(* Logix 5000 project; controller STAT 1756-L72 rev 20.12; software revision 20.04; part 33 of 34 *)
(* tags used below, declared in another part *)
   B3 : DINT[50];
   F8 : REAL[200];
   I1_000_Bit00 : ALIAS FOR stock:1:I.Point_0;   // disjoncteur algemeen
   I1_000_Bit01 : ALIAS FOR stock:1:I.Point_1;   // alim rechauffeur1
   I1_000_Bit02 : ALIAS FOR stock:1:I.Point_2;   // alim rechauffeur2
   I1_000_Bit03 : ALIAS FOR stock:1:I.Point_3;   // alim rechauffeur 3
   I1_000_Bit04 : ALIAS FOR stock:1:I.Point_4;   // alim rechauffeur 4
   I1_000_Bit05 : ALIAS FOR stock:1:I.Point_5;   // alim rechauffeur 5
   I1_000_Bit06 : ALIAS FOR stock:1:I.Point_6;   // protection pompesoude
   I1_000_Bit07 : ALIAS FOR stock:1:I.Point_7;   // protection pmp 2 acide
   I1_000_Bit08 : ALIAS FOR stock:1:I.Point_8;   // protection pmp acide
   I1_000_Bit15 : ALIAS FOR stock:1:I.Point_15;   // arret urgence
   I1_001_Bit09 : ALIAS FOR stock:1:I.Point_25;   // select.pmp soude sur drive
   I1_001_Bit11 : ALIAS FOR stock:1:I.Point_27;   // fault drivepmp soude
   I2_000_Bit00 : ALIAS FOR stock:2:I.Point_0;   // detection fuite soud
   I2_000_Bit01 : ALIAS FOR stock:2:I.Point_1;   // detection fuite acid
   I2_000_Bit02 : ALIAS FOR stock:2:I.Point_2;   // detection fuite mazo
   I2_000_Bit03 : ALIAS FOR stock:2:I.Point_3;   // wegskraan soude open
   I2_000_Bit04 : ALIAS FOR stock:2:I.Point_4;   // wegskraan soude dich
   I2_000_Bit07 : ALIAS FOR stock:2:I.Point_7;   // overfill stockagesoude
   I2_000_Bit08 : ALIAS FOR stock:2:I.Point_8;   // detection acideencuvement
   I2_000_Bit09 : ALIAS FOR stock:2:I.Point_9;   // detection soudeencuvement
   I2_000_Bit10 : ALIAS FOR stock:2:I.Point_10;   // fv vannesecuriteacide OUVERT
   I2_000_Bit11 : ALIAS FOR stock:2:I.Point_11;   // fv vannesecuriteacide FERME
   I2_001_Bit00 : ALIAS FOR stock:2:I.Point_16;   // NAOHL1 VA4FC O
   I2_001_Bit01 : ALIAS FOR stock:2:I.Point_17;   // NAOHL1 VA4FC F
   I2_001_Bit02 : ALIAS FOR stock:2:I.Point_18;   // NAOHL2 VA4FC O
   I2_001_Bit03 : ALIAS FOR stock:2:I.Point_19;   // NAOHL2 VA4FC O
   I2_001_Bit15 : ALIAS FOR stock:2:I.Point_31;   // pulse 0.1L passé
   N20 : DINT[100];
   N7 : DINT[255];
   O3_000_Bit00 : ALIAS FOR stock:3:O.Point_0;   // pompe soude
   O3_000_Bit08 : ALIAS FOR stock:3:O.Point_8;   // vanne soude
   O3_000_Bit09 : ALIAS FOR stock:3:O.Point_9;   // vannesecuriteacide
   O3_001_Bit11 : ALIAS FOR stock:3:O.Point_27;   // L1 VA4
   O3_001_Bit12 : ALIAS FOR stock:3:O.Point_28;   // NAOHL2 VA4
   T4 : TIMER[50];
   DateTime : DINT[7];   // DINT array tag for retrieve wallclock time through GSV created during conversion
   dmd_h2so4_ibt_ok : BOOL;
   dmd_soude_ibt_ok : BOOL;
   h2so4_ibt_finit : BOOL;
   I19_001_Bit05 : ALIAS FOR I19[1].5;   // vanne acide de stock fermee
   I19_001_Bit06 : ALIAS FOR I19[1].6;   // vanne acide de stock ouverte
   L1_stat : DINT[20];
   L2_STAT : DINT[20];
   L3_STAT : DINT[20];
   lancystock1 : DINT;
   lastmonth_h2so4_L1 : DINT;
   lastmonth_h2so4_L2 : DINT;
   lastmonth_h2so4_L3 : DINT;
   lastmonth_h2so4_L4 : DINT;
   lastmonth_h2so4_stat : REAL;
   lastmonth_naoh_L1 : DINT;
   lastmonth_naoh_L2 : DINT;
   lastmonth_naoh_L3 : DINT;
   lastmonth_naoh_L4 : DINT;
   lastmonth_naoh_stat : DINT;
   memo_flow_l1 : REAL;
   memo_flow_l2 : REAL;
   memo_flow_l3 : REAL;
   MW1 : BOOL;
   N : INT[255];
   O16_000_Bit03 : ALIAS FOR O16[0].3;
   ONS1 : DINT;
   passage_jourmois : BOOL;
   s_dmd_acid_ibt : DINT;
   S_dmd_naoh_ibt : REAL;
   s_lastmonth_tot_h2o_l1 : REAL;
   s_lastmonth_tot_h2o_l2 : REAL;
   s_lastmonth_tot_h2o_l3 : REAL;
   S_stock_v_h2so4_f : BOOL;
   S_stock_v_h2so4_o : BOOL;
   stat_L1 : DINT[20];
   STAT_L2 : DINT[20];
   STAT_L3 : DINT[20];
   stocklancy1 : DINT;
   stocklancy2 : DINT;
   tot_h2so4_stat : REAL;
   water_flow_to_l1 : REAL;
   water_flow_to_l2 : REAL;
   water_flow_to_l3 : REAL;
(* stock, continued *)

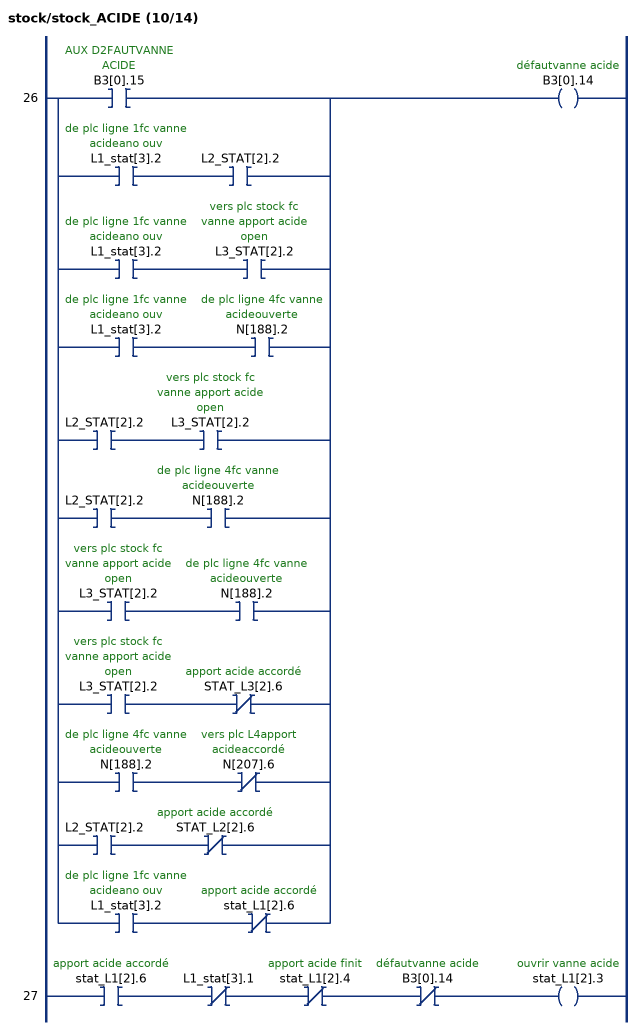
   [picture p674: stock/stock_ACIDE rungs 26-27]
   26: [XIC(B3[0].15) ,XIC(L1_stat[3].2) XIC(L2_STAT[2].2) ,XIC(L1_stat[3].2) XIC(L3_STAT[2].2) ,XIC(L1_stat[3].2) XIC(N[188].2) ,XIC(L2_STAT[2].2) XIC(L3_STAT[2].2) ,XIC(L2_STAT[2].2) XIC(N[188].2) ,XIC(L3_STAT[2].2) XIC(N[188].2) ,XIC(L3_STAT[2].2) XIO(STAT_L3[2].6) ,XIC(N[188].2) XIO(N[207].6) ,XIC(L2_STAT[2].2) XIO(STAT_L2[2].6) ,XIC(L1_stat[3].2) XIO(stat_L1[2].6) ]OTE(B3[0].14);
   27: XIC(stat_L1[2].6)XIO(L1_stat[3].1)XIO(stat_L1[2].4)XIO(B3[0].14)OTE(stat_L1[2].3);
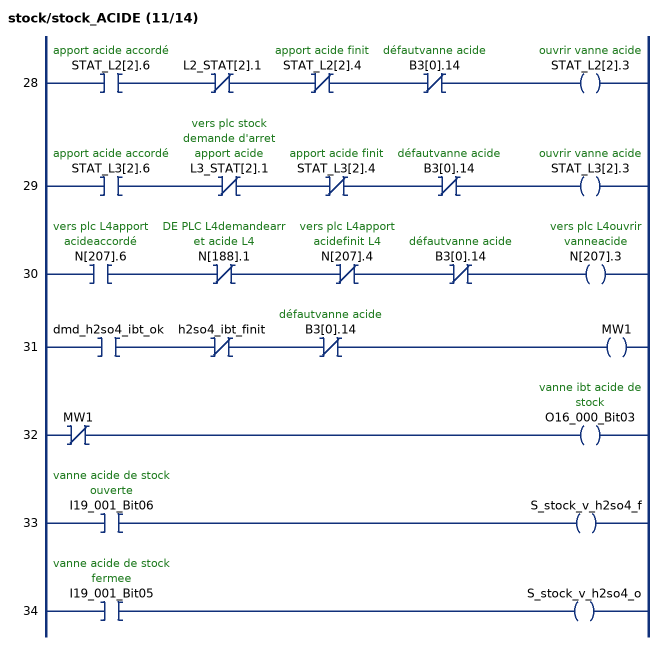
   28: XIC(STAT_L2[2].6)XIO(L2_STAT[2].1)XIO(STAT_L2[2].4)XIO(B3[0].14)OTE(STAT_L2[2].3);
   29: XIC(STAT_L3[2].6)XIO(L3_STAT[2].1)XIO(STAT_L3[2].4)XIO(B3[0].14)OTE(STAT_L3[2].3);
   30: XIC(N[207].6)XIO(N[188].1)XIO(N[207].4)XIO(B3[0].14)OTE(N[207].3);
   31: XIC(dmd_h2so4_ibt_ok)XIO(h2so4_ibt_finit)XIO(B3[0].14)OTE(MW1);
   32: XIO(MW1)OTE(O16_000_Bit03);
   33: XIC(I19_001_Bit06)OTE(S_stock_v_h2so4_f);
   34: XIC(I19_001_Bit05)OTE(S_stock_v_h2so4_o);
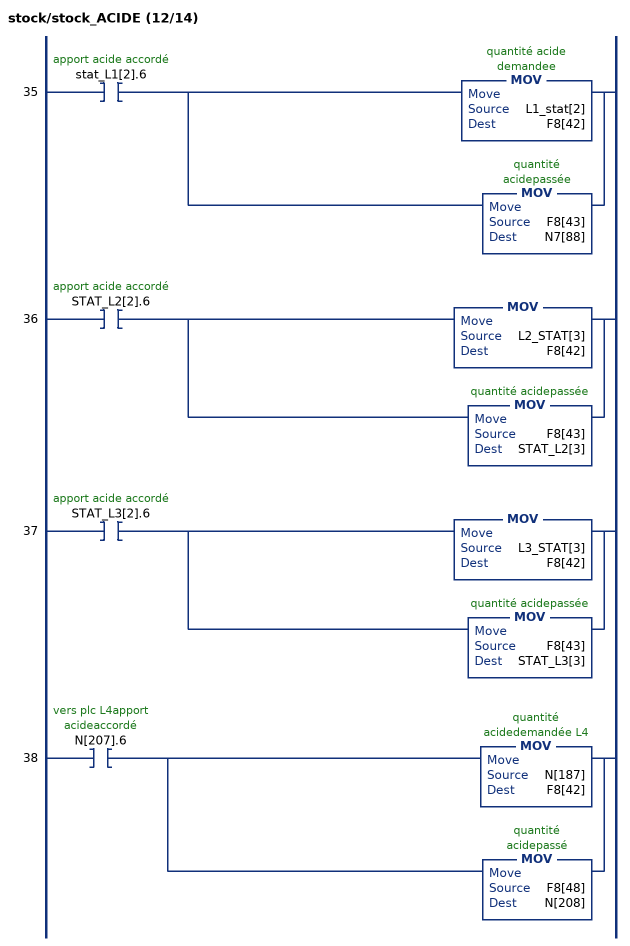
   35: XIC(stat_L1[2].6)[MOV(L1_stat[2],F8[42]) ,MOV(F8[43],N7[88]) ];
   36: XIC(STAT_L2[2].6)[MOV(L2_STAT[3],F8[42]) ,MOV(F8[43],STAT_L2[3]) ];
   37: XIC(STAT_L3[2].6)[MOV(L3_STAT[3],F8[42]) ,MOV(F8[43],STAT_L3[3]) ];
   38: XIC(N[207].6)[MOV(N[187],F8[42]) ,MOV(F8[48],N[208]) ];
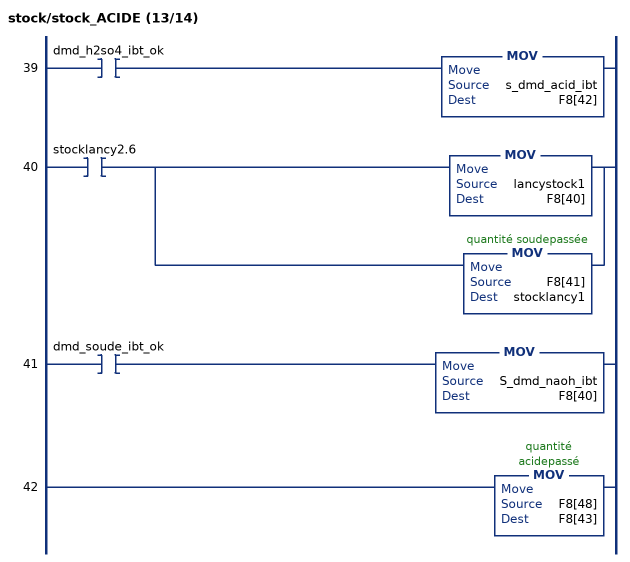
   39: XIC(dmd_h2so4_ibt_ok)MOV(s_dmd_acid_ibt,F8[42]);
   40: XIC(stocklancy2.6)[MOV(lancystock1,F8[40]) ,MOV(F8[41],stocklancy1) ];
   41: XIC(dmd_soude_ibt_ok)MOV(S_dmd_naoh_ibt,F8[40]);
   42: MOV(F8[48],F8[43]);
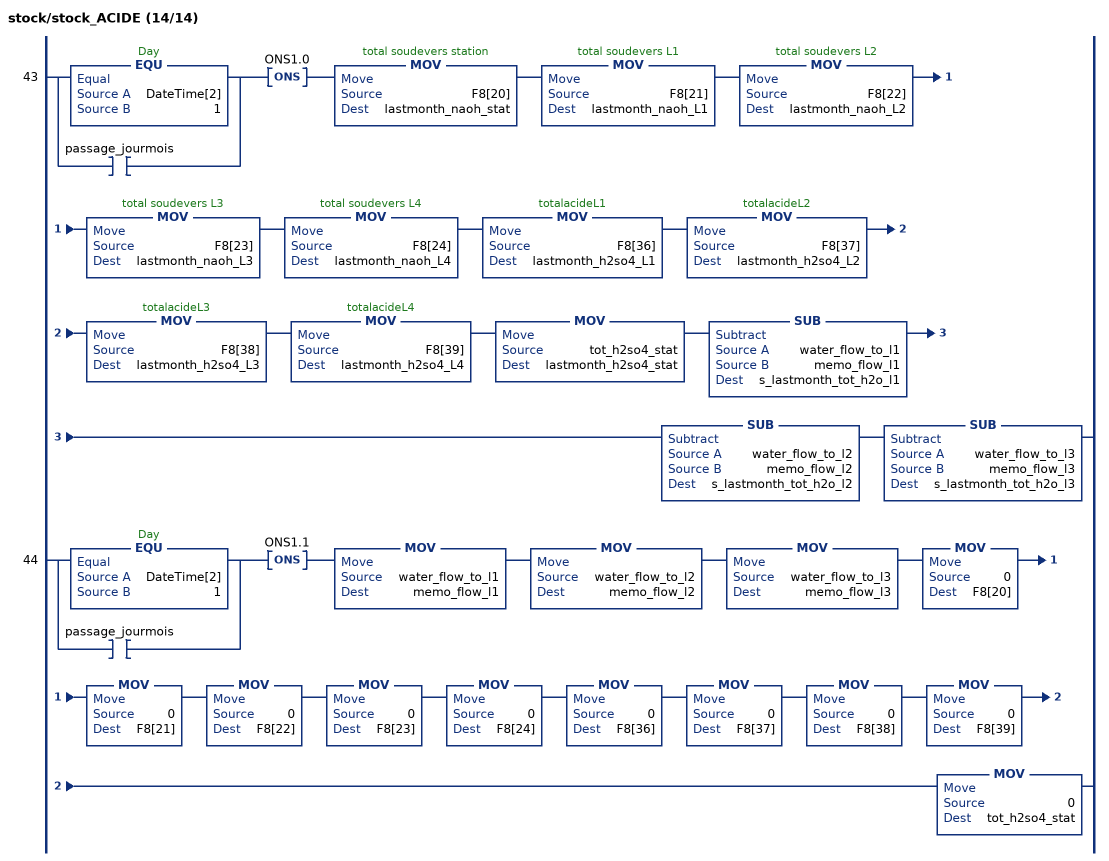
   43: [EQU(DateTime[2],1) ,XIC(passage_jourmois) ]ONS(ONS1.0)MOV(F8[20],lastmonth_naoh_stat)MOV(F8[21],lastmonth_naoh_L1)MOV(F8[22],lastmonth_naoh_L2)MOV(F8[23],lastmonth_naoh_L3)MOV(F8[24],lastmonth_naoh_L4)MOV(F8[36],lastmonth_h2so4_L1)MOV(F8[37],lastmonth_h2so4_L2)MOV(F8[38],lastmonth_h2so4_L3)MOV(F8[39],lastmonth_h2so4_L4)MOV(tot_h2so4_stat,lastmonth_h2so4_stat)SUB(water_flow_to_l1,memo_flow_l1,s_lastmonth_tot_h2o_l1)SUB(water_flow_to_l2,memo_flow_l2,s_lastmonth_tot_h2o_l2)SUB(water_flow_to_l3,memo_flow_l3,s_lastmonth_tot_h2o_l3);
   44: [EQU(DateTime[2],1) ,XIC(passage_jourmois) ]ONS(ONS1.1)MOV(water_flow_to_l1,memo_flow_l1)MOV(water_flow_to_l2,memo_flow_l2)MOV(water_flow_to_l3,memo_flow_l3)MOV(0,F8[20])MOV(0,F8[21])MOV(0,F8[22])MOV(0,F8[23])MOV(0,F8[24])MOV(0,F8[36])MOV(0,F8[37])MOV(0,F8[38])MOV(0,F8[39])MOV(0,tot_h2so4_stat);
END_ROUTINE

ROUTINE stock_ALARMING   (* ladder *)
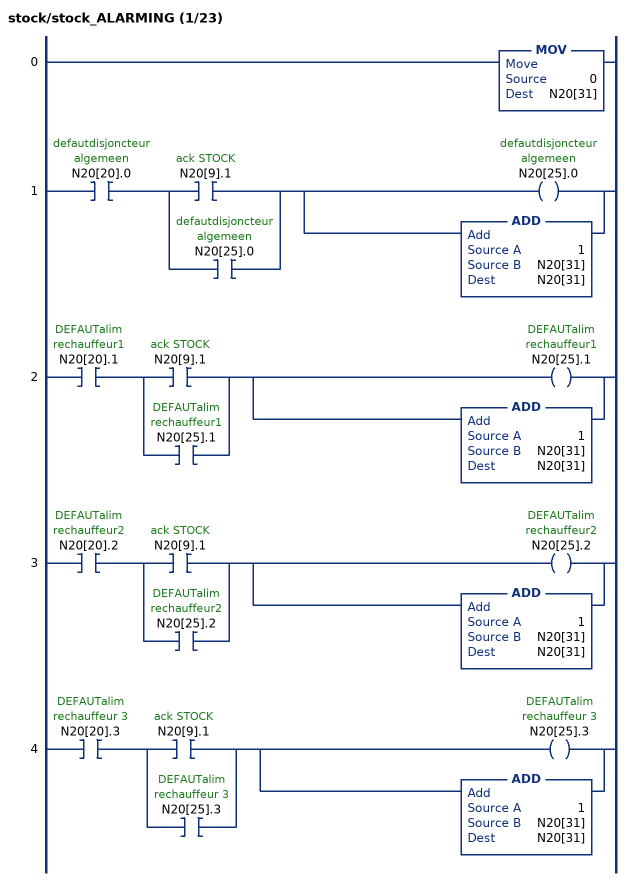
   0: MOV(0,N20[31]);
   1: XIC(N20[20].0)[XIC(N20[9].1) ,XIC(N20[25].0) ][OTE(N20[25].0) ,ADD(1,N20[31],N20[31]) ];
   2: XIC(N20[20].1)[XIC(N20[9].1) ,XIC(N20[25].1) ][OTE(N20[25].1) ,ADD(1,N20[31],N20[31]) ];
   3: XIC(N20[20].2)[XIC(N20[9].1) ,XIC(N20[25].2) ][OTE(N20[25].2) ,ADD(1,N20[31],N20[31]) ];
   4: XIC(N20[20].3)[XIC(N20[9].1) ,XIC(N20[25].3) ][OTE(N20[25].3) ,ADD(1,N20[31],N20[31]) ];
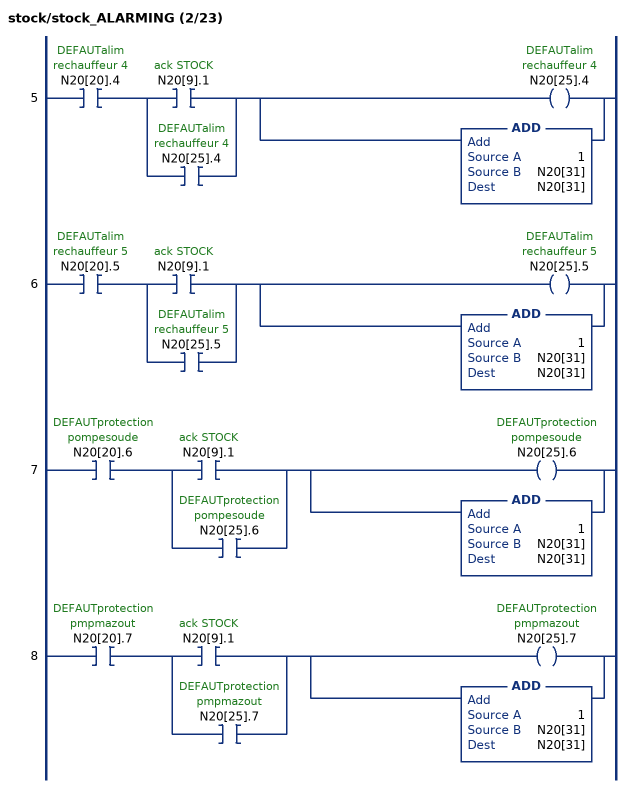
   5: XIC(N20[20].4)[XIC(N20[9].1) ,XIC(N20[25].4) ][OTE(N20[25].4) ,ADD(1,N20[31],N20[31]) ];
   6: XIC(N20[20].5)[XIC(N20[9].1) ,XIC(N20[25].5) ][OTE(N20[25].5) ,ADD(1,N20[31],N20[31]) ];
   7: XIC(N20[20].6)[XIC(N20[9].1) ,XIC(N20[25].6) ][OTE(N20[25].6) ,ADD(1,N20[31],N20[31]) ];
   8: XIC(N20[20].7)[XIC(N20[9].1) ,XIC(N20[25].7) ][OTE(N20[25].7) ,ADD(1,N20[31],N20[31]) ];
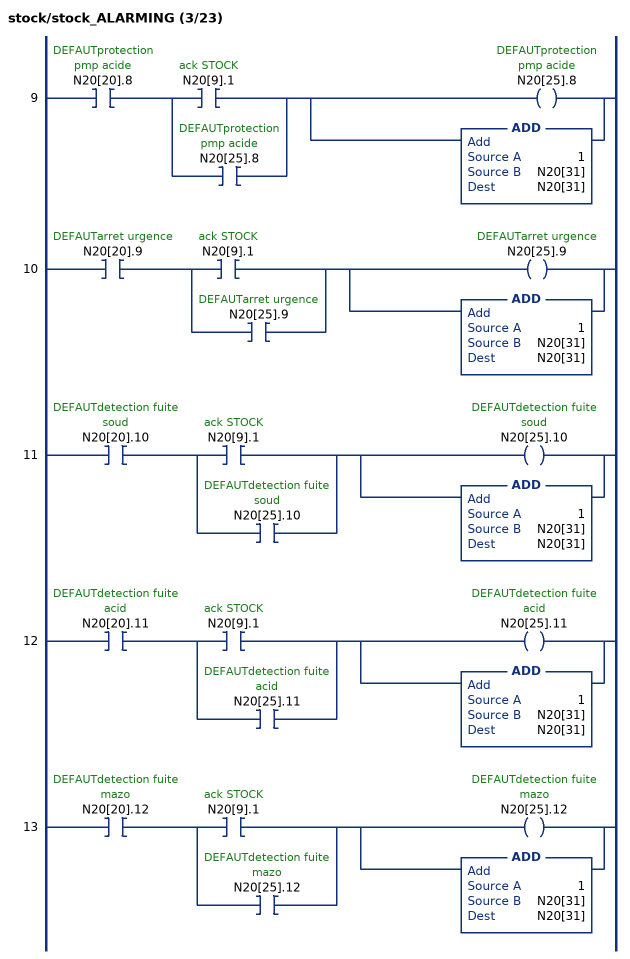
   9: XIC(N20[20].8)[XIC(N20[9].1) ,XIC(N20[25].8) ][OTE(N20[25].8) ,ADD(1,N20[31],N20[31]) ];
   10: XIC(N20[20].9)[XIC(N20[9].1) ,XIC(N20[25].9) ][OTE(N20[25].9) ,ADD(1,N20[31],N20[31]) ];
   11: XIC(N20[20].10)[XIC(N20[9].1) ,XIC(N20[25].10) ][OTE(N20[25].10) ,ADD(1,N20[31],N20[31]) ];
   12: XIC(N20[20].11)[XIC(N20[9].1) ,XIC(N20[25].11) ][OTE(N20[25].11) ,ADD(1,N20[31],N20[31]) ];
   13: XIC(N20[20].12)[XIC(N20[9].1) ,XIC(N20[25].12) ][OTE(N20[25].12) ,ADD(1,N20[31],N20[31]) ];
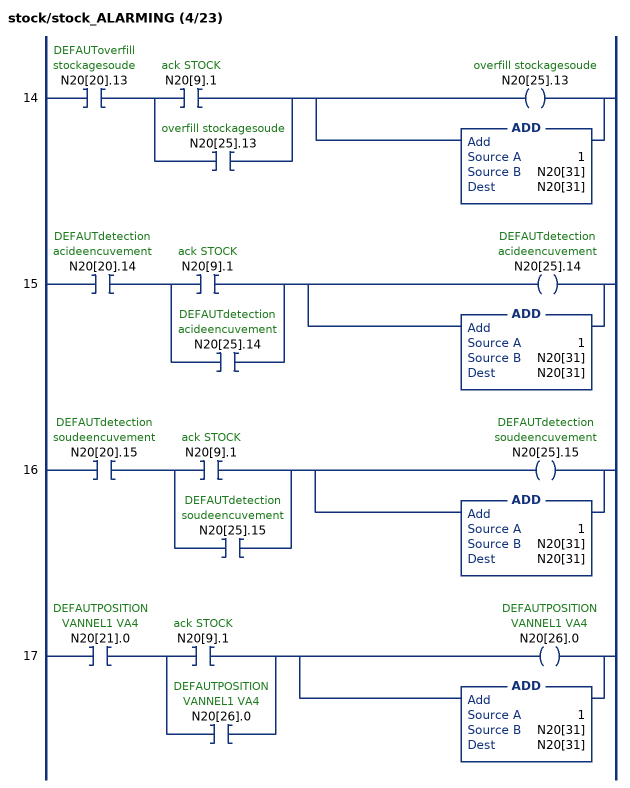
   14: XIC(N20[20].13)[XIC(N20[9].1) ,XIC(N20[25].13) ][OTE(N20[25].13) ,ADD(1,N20[31],N20[31]) ];
   15: XIC(N20[20].14)[XIC(N20[9].1) ,XIC(N20[25].14) ][OTE(N20[25].14) ,ADD(1,N20[31],N20[31]) ];
   16: XIC(N20[20].15)[XIC(N20[9].1) ,XIC(N20[25].15) ][OTE(N20[25].15) ,ADD(1,N20[31],N20[31]) ];
   17: XIC(N20[21].0)[XIC(N20[9].1) ,XIC(N20[26].0) ][OTE(N20[26].0) ,ADD(1,N20[31],N20[31]) ];
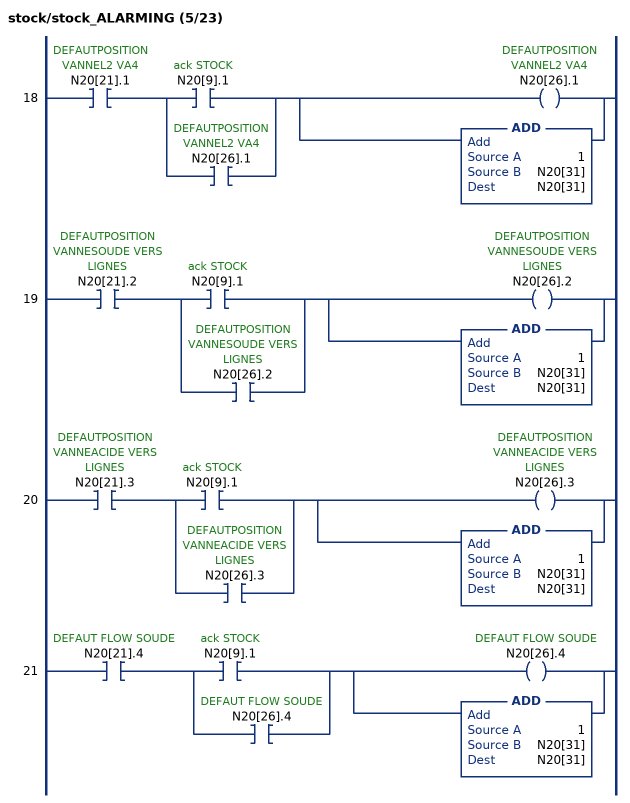
   18: XIC(N20[21].1)[XIC(N20[9].1) ,XIC(N20[26].1) ][OTE(N20[26].1) ,ADD(1,N20[31],N20[31]) ];
   19: XIC(N20[21].2)[XIC(N20[9].1) ,XIC(N20[26].2) ][OTE(N20[26].2) ,ADD(1,N20[31],N20[31]) ];
   20: XIC(N20[21].3)[XIC(N20[9].1) ,XIC(N20[26].3) ][OTE(N20[26].3) ,ADD(1,N20[31],N20[31]) ];
   21: XIC(N20[21].4)[XIC(N20[9].1) ,XIC(N20[26].4) ][OTE(N20[26].4) ,ADD(1,N20[31],N20[31]) ];
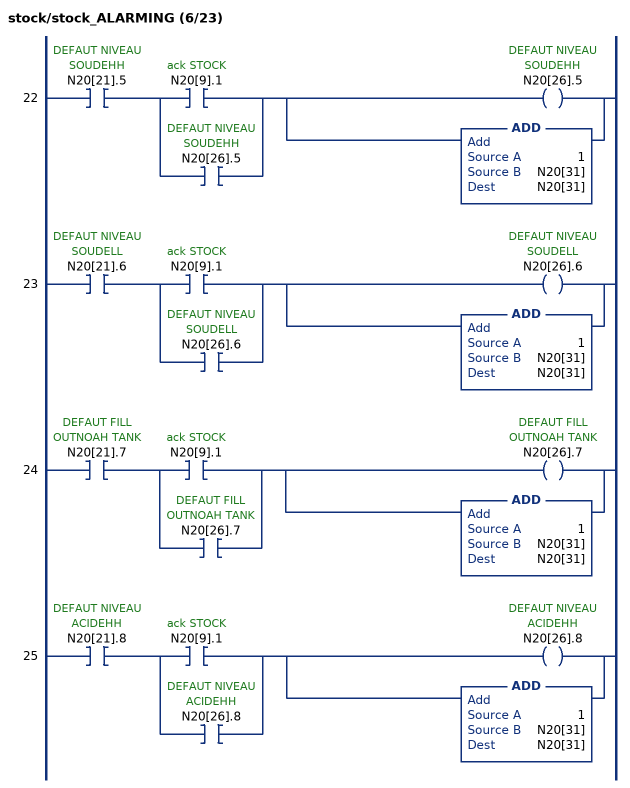
   22: XIC(N20[21].5)[XIC(N20[9].1) ,XIC(N20[26].5) ][OTE(N20[26].5) ,ADD(1,N20[31],N20[31]) ];
   23: XIC(N20[21].6)[XIC(N20[9].1) ,XIC(N20[26].6) ][OTE(N20[26].6) ,ADD(1,N20[31],N20[31]) ];
   24: XIC(N20[21].7)[XIC(N20[9].1) ,XIC(N20[26].7) ][OTE(N20[26].7) ,ADD(1,N20[31],N20[31]) ];
   25: XIC(N20[21].8)[XIC(N20[9].1) ,XIC(N20[26].8) ][OTE(N20[26].8) ,ADD(1,N20[31],N20[31]) ];
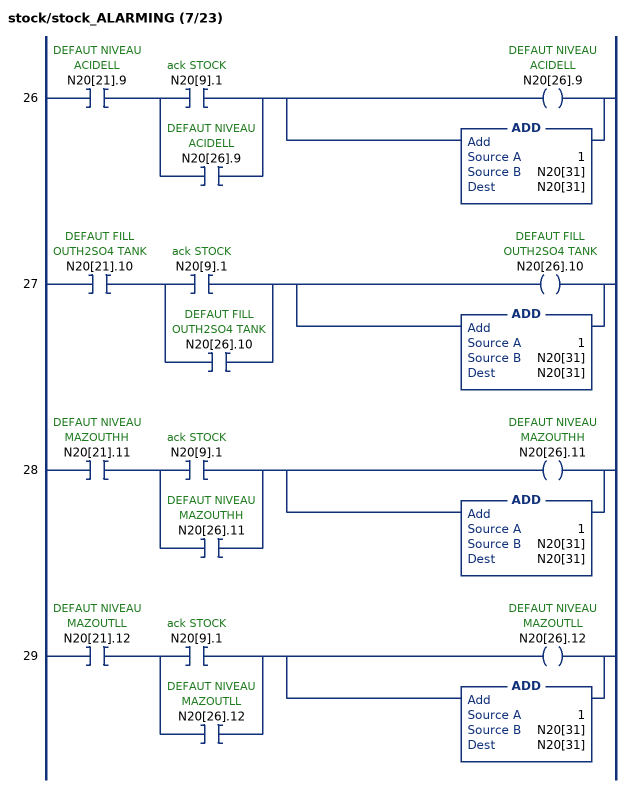
   26: XIC(N20[21].9)[XIC(N20[9].1) ,XIC(N20[26].9) ][OTE(N20[26].9) ,ADD(1,N20[31],N20[31]) ];
   27: XIC(N20[21].10)[XIC(N20[9].1) ,XIC(N20[26].10) ][OTE(N20[26].10) ,ADD(1,N20[31],N20[31]) ];
   28: XIC(N20[21].11)[XIC(N20[9].1) ,XIC(N20[26].11) ][OTE(N20[26].11) ,ADD(1,N20[31],N20[31]) ];
   29: XIC(N20[21].12)[XIC(N20[9].1) ,XIC(N20[26].12) ][OTE(N20[26].12) ,ADD(1,N20[31],N20[31]) ];
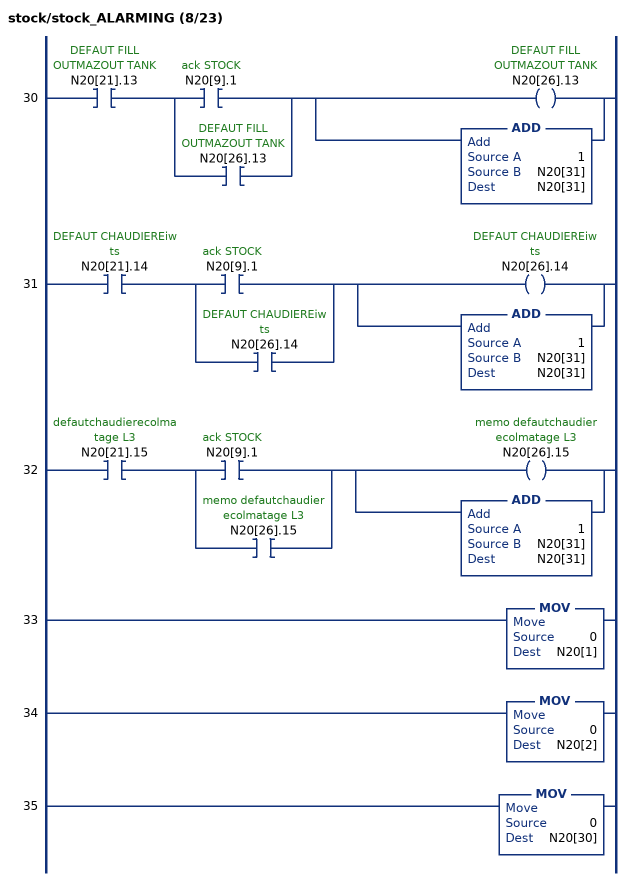
   30: XIC(N20[21].13)[XIC(N20[9].1) ,XIC(N20[26].13) ][OTE(N20[26].13) ,ADD(1,N20[31],N20[31]) ];
   31: XIC(N20[21].14)[XIC(N20[9].1) ,XIC(N20[26].14) ][OTE(N20[26].14) ,ADD(1,N20[31],N20[31]) ];
   32: XIC(N20[21].15)[XIC(N20[9].1) ,XIC(N20[26].15) ][OTE(N20[26].15) ,ADD(1,N20[31],N20[31]) ];
   33: MOV(0,N20[1]);
   34: MOV(0,N20[2]);
   35: MOV(0,N20[30]);
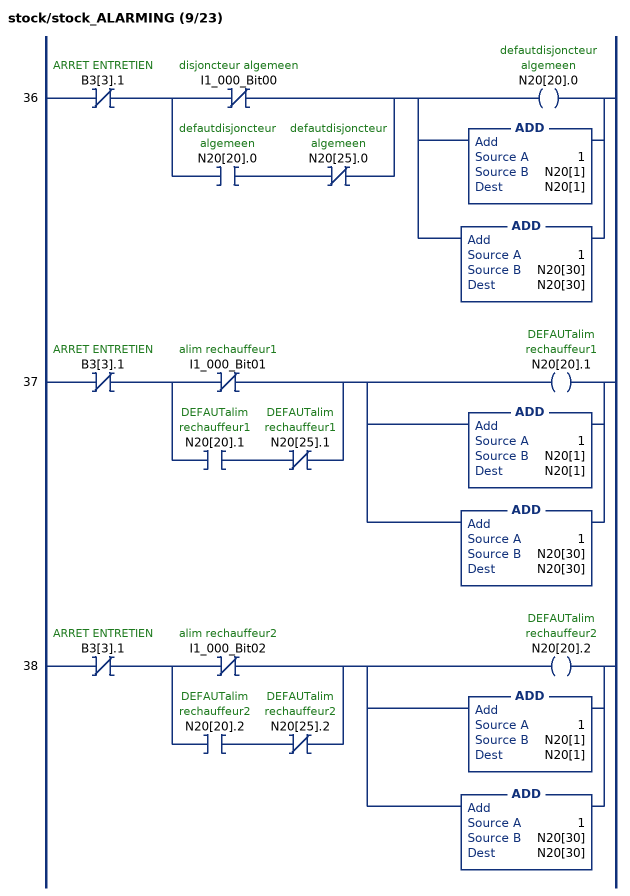
   36: XIO(B3[3].1)[XIO(I1_000_Bit00) ,XIC(N20[20].0) XIO(N20[25].0) ][OTE(N20[20].0) ,ADD(1,N20[1],N20[1]) ,ADD(1,N20[30],N20[30]) ];
   37: XIO(B3[3].1)[XIO(I1_000_Bit01) ,XIC(N20[20].1) XIO(N20[25].1) ][OTE(N20[20].1) ,ADD(1,N20[1],N20[1]) ,ADD(1,N20[30],N20[30]) ];
   38: XIO(B3[3].1)[XIO(I1_000_Bit02) ,XIC(N20[20].2) XIO(N20[25].2) ][OTE(N20[20].2) ,ADD(1,N20[1],N20[1]) ,ADD(1,N20[30],N20[30]) ];
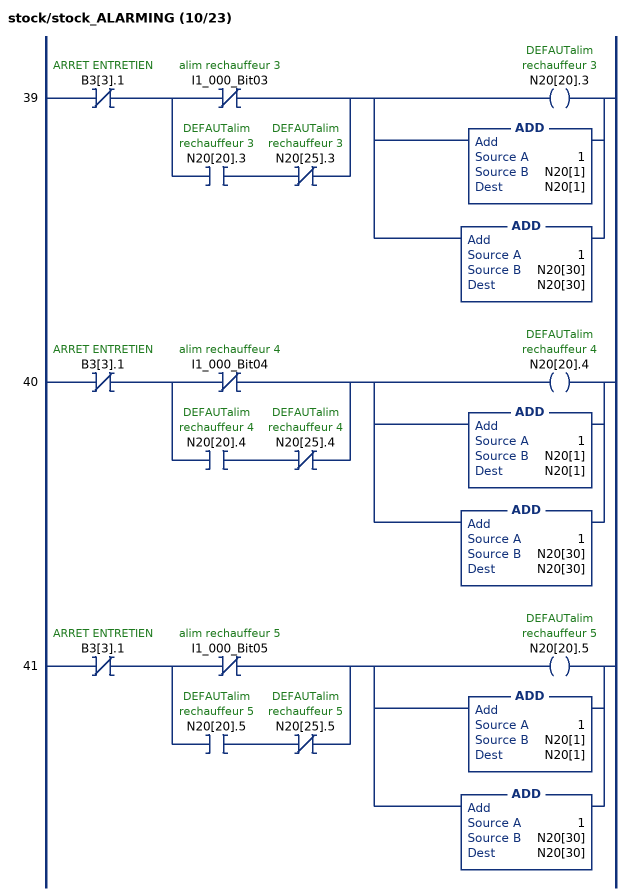
   39: XIO(B3[3].1)[XIO(I1_000_Bit03) ,XIC(N20[20].3) XIO(N20[25].3) ][OTE(N20[20].3) ,ADD(1,N20[1],N20[1]) ,ADD(1,N20[30],N20[30]) ];
   40: XIO(B3[3].1)[XIO(I1_000_Bit04) ,XIC(N20[20].4) XIO(N20[25].4) ][OTE(N20[20].4) ,ADD(1,N20[1],N20[1]) ,ADD(1,N20[30],N20[30]) ];
   41: XIO(B3[3].1)[XIO(I1_000_Bit05) ,XIC(N20[20].5) XIO(N20[25].5) ][OTE(N20[20].5) ,ADD(1,N20[1],N20[1]) ,ADD(1,N20[30],N20[30]) ];
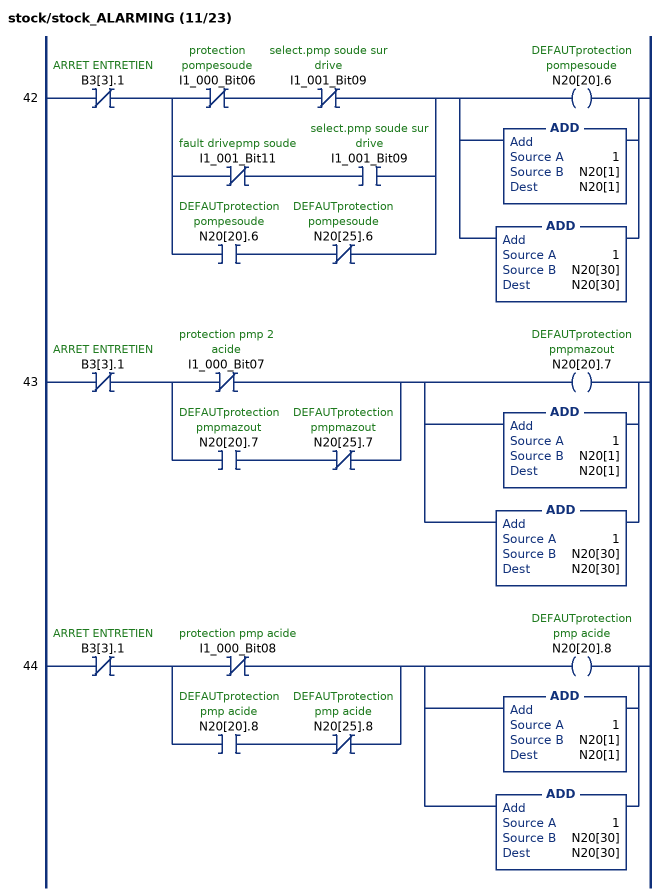
   42: XIO(B3[3].1)[XIO(I1_000_Bit06) XIO(I1_001_Bit09) ,XIO(I1_001_Bit11) XIC(I1_001_Bit09) ,XIC(N20[20].6) XIO(N20[25].6) ][OTE(N20[20].6) ,ADD(1,N20[1],N20[1]) ,ADD(1,N20[30],N20[30]) ];
   43: XIO(B3[3].1)[XIO(I1_000_Bit07) ,XIC(N20[20].7) XIO(N20[25].7) ][OTE(N20[20].7) ,ADD(1,N20[1],N20[1]) ,ADD(1,N20[30],N20[30]) ];
   44: XIO(B3[3].1)[XIO(I1_000_Bit08) ,XIC(N20[20].8) XIO(N20[25].8) ][OTE(N20[20].8) ,ADD(1,N20[1],N20[1]) ,ADD(1,N20[30],N20[30]) ];
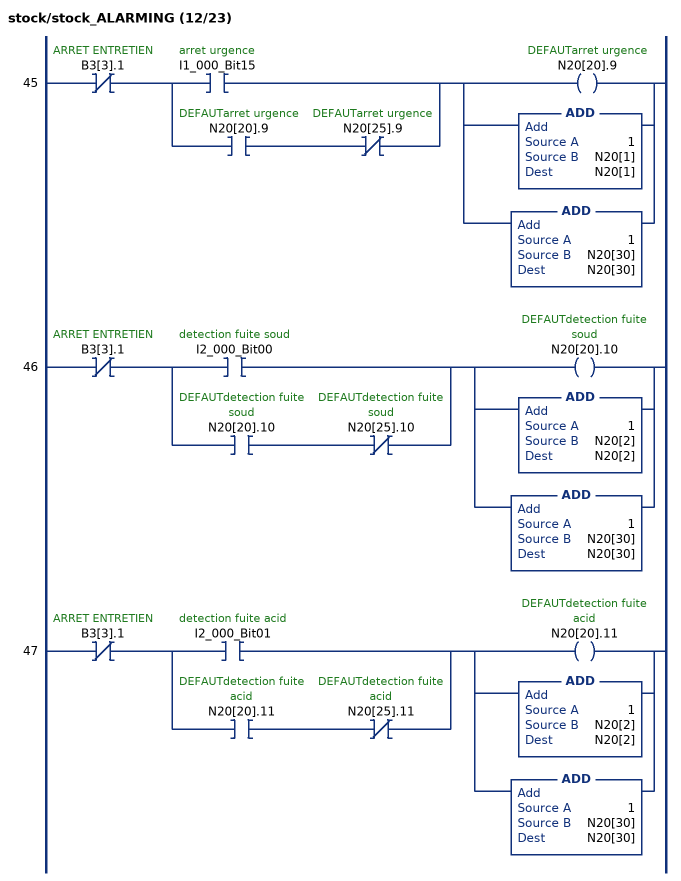
   45: XIO(B3[3].1)[XIC(I1_000_Bit15) ,XIC(N20[20].9) XIO(N20[25].9) ][OTE(N20[20].9) ,ADD(1,N20[1],N20[1]) ,ADD(1,N20[30],N20[30]) ];
   46: XIO(B3[3].1)[XIC(I2_000_Bit00) ,XIC(N20[20].10) XIO(N20[25].10) ][OTE(N20[20].10) ,ADD(1,N20[2],N20[2]) ,ADD(1,N20[30],N20[30]) ];
   47: XIO(B3[3].1)[XIC(I2_000_Bit01) ,XIC(N20[20].11) XIO(N20[25].11) ][OTE(N20[20].11) ,ADD(1,N20[2],N20[2]) ,ADD(1,N20[30],N20[30]) ];
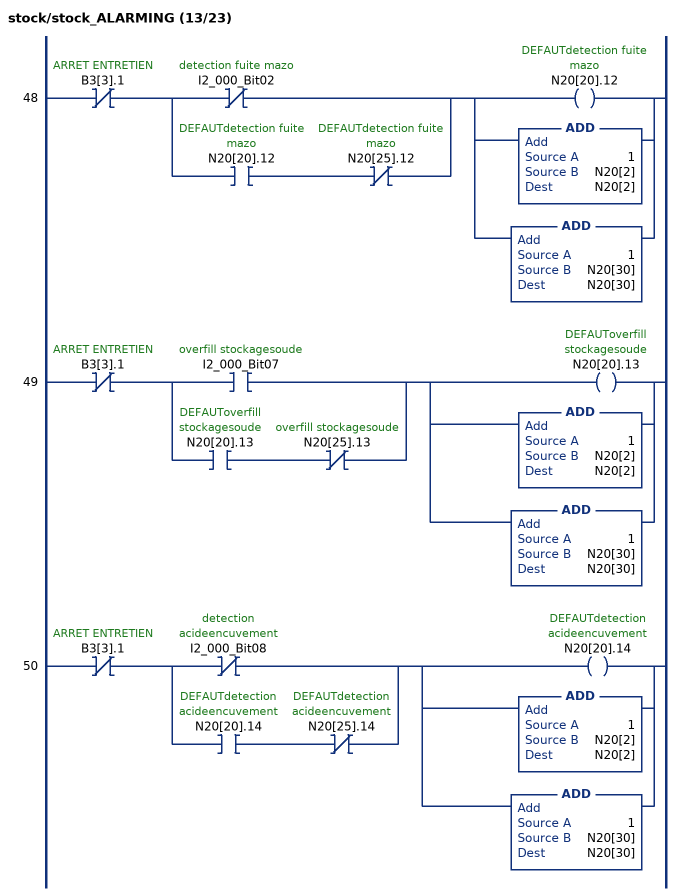
   48: XIO(B3[3].1)[XIO(I2_000_Bit02) ,XIC(N20[20].12) XIO(N20[25].12) ][OTE(N20[20].12) ,ADD(1,N20[2],N20[2]) ,ADD(1,N20[30],N20[30]) ];
   49: XIO(B3[3].1)[XIC(I2_000_Bit07) ,XIC(N20[20].13) XIO(N20[25].13) ][OTE(N20[20].13) ,ADD(1,N20[2],N20[2]) ,ADD(1,N20[30],N20[30]) ];
   50: XIO(B3[3].1)[XIO(I2_000_Bit08) ,XIC(N20[20].14) XIO(N20[25].14) ][OTE(N20[20].14) ,ADD(1,N20[2],N20[2]) ,ADD(1,N20[30],N20[30]) ];
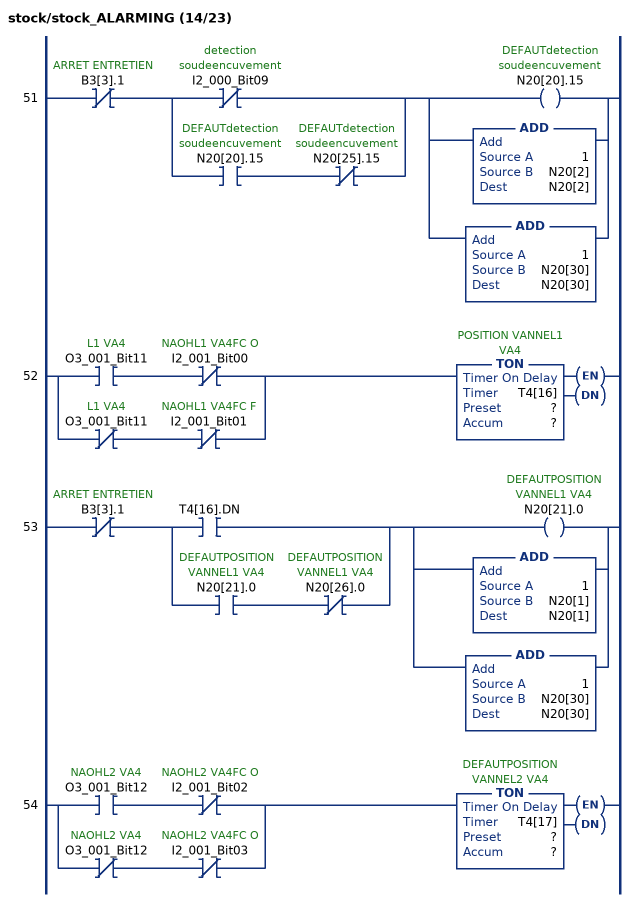
   51: XIO(B3[3].1)[XIO(I2_000_Bit09) ,XIC(N20[20].15) XIO(N20[25].15) ][OTE(N20[20].15) ,ADD(1,N20[2],N20[2]) ,ADD(1,N20[30],N20[30]) ];
   52: [XIC(O3_001_Bit11) XIO(I2_001_Bit00) ,XIO(O3_001_Bit11) XIO(I2_001_Bit01) ]TON(T4[16],?,?);
   53: XIO(B3[3].1)[XIC(T4[16].DN) ,XIC(N20[21].0) XIO(N20[26].0) ][OTE(N20[21].0) ,ADD(1,N20[1],N20[1]) ,ADD(1,N20[30],N20[30]) ];
   54: [XIC(O3_001_Bit12) XIO(I2_001_Bit02) ,XIO(O3_001_Bit12) XIO(I2_001_Bit03) ]TON(T4[17],?,?);
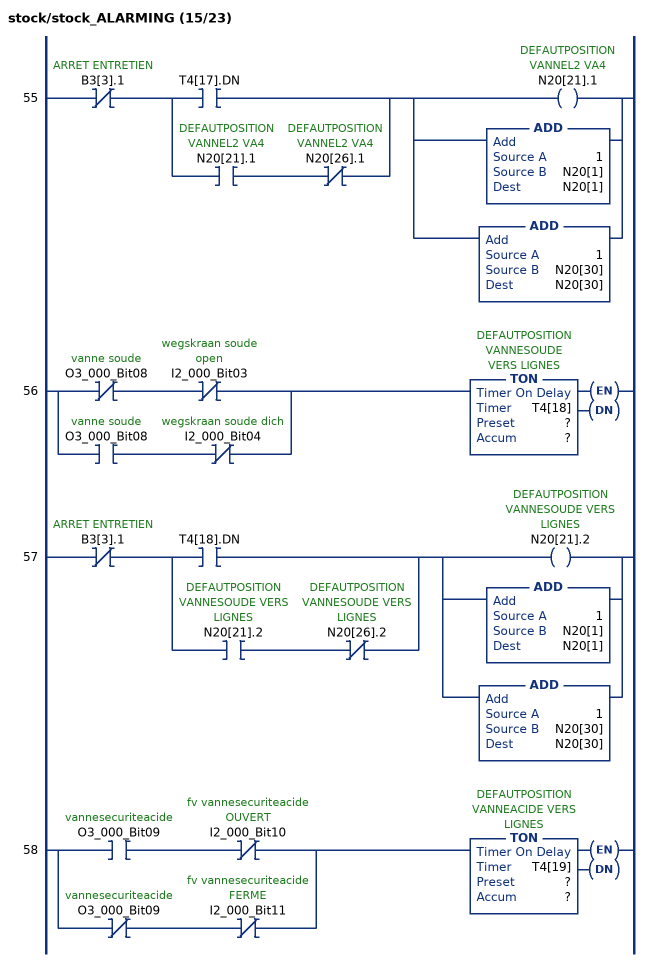
   55: XIO(B3[3].1)[XIC(T4[17].DN) ,XIC(N20[21].1) XIO(N20[26].1) ][OTE(N20[21].1) ,ADD(1,N20[1],N20[1]) ,ADD(1,N20[30],N20[30]) ];
   56: [XIO(O3_000_Bit08) XIO(I2_000_Bit03) ,XIC(O3_000_Bit08) XIO(I2_000_Bit04) ]TON(T4[18],?,?);
   57: XIO(B3[3].1)[XIC(T4[18].DN) ,XIC(N20[21].2) XIO(N20[26].2) ][OTE(N20[21].2) ,ADD(1,N20[1],N20[1]) ,ADD(1,N20[30],N20[30]) ];
   58: [XIC(O3_000_Bit09) XIO(I2_000_Bit10) ,XIO(O3_000_Bit09) XIO(I2_000_Bit11) ]TON(T4[19],?,?);
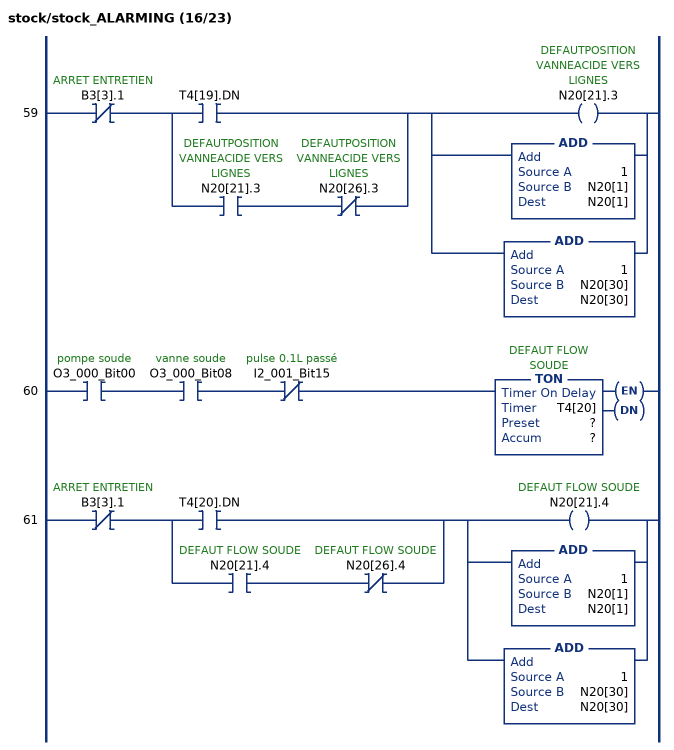
   59: XIO(B3[3].1)[XIC(T4[19].DN) ,XIC(N20[21].3) XIO(N20[26].3) ][OTE(N20[21].3) ,ADD(1,N20[1],N20[1]) ,ADD(1,N20[30],N20[30]) ];
   60: XIC(O3_000_Bit00)XIC(O3_000_Bit08)XIO(I2_001_Bit15)TON(T4[20],?,?);
   61: XIO(B3[3].1)[XIC(T4[20].DN) ,XIC(N20[21].4) XIO(N20[26].4) ][OTE(N20[21].4) ,ADD(1,N20[1],N20[1]) ,ADD(1,N20[30],N20[30]) ];
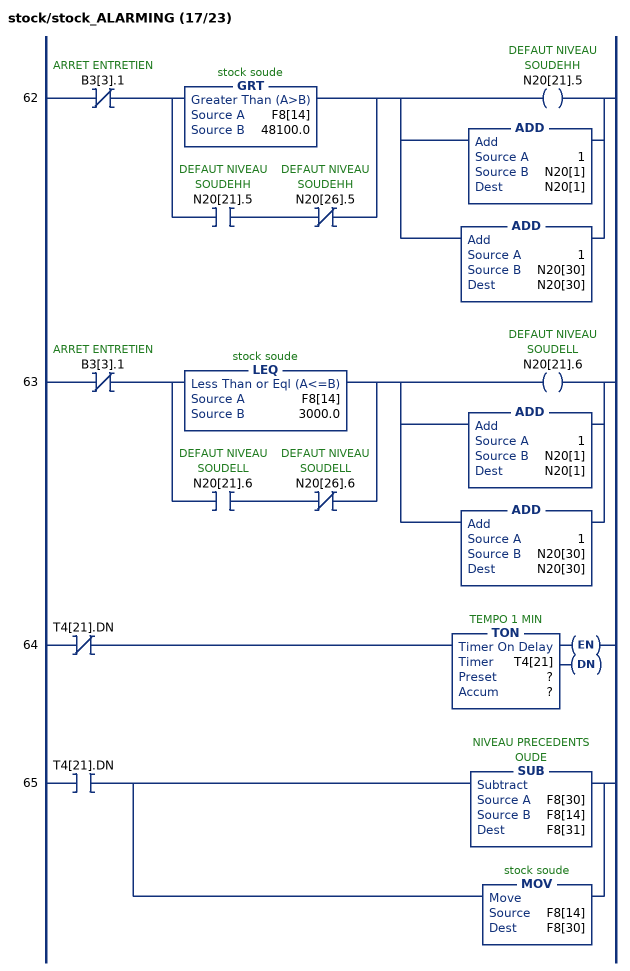
   62: XIO(B3[3].1)[GRT(F8[14],48100.0) ,XIC(N20[21].5) XIO(N20[26].5) ][OTE(N20[21].5) ,ADD(1,N20[1],N20[1]) ,ADD(1,N20[30],N20[30]) ];
   63: XIO(B3[3].1)[LEQ(F8[14],3000.0) ,XIC(N20[21].6) XIO(N20[26].6) ][OTE(N20[21].6) ,ADD(1,N20[1],N20[1]) ,ADD(1,N20[30],N20[30]) ];
   64: XIO(T4[21].DN)TON(T4[21],?,?);
   65: XIC(T4[21].DN)[SUB(F8[30],F8[14],F8[31]) ,MOV(F8[14],F8[30]) ];
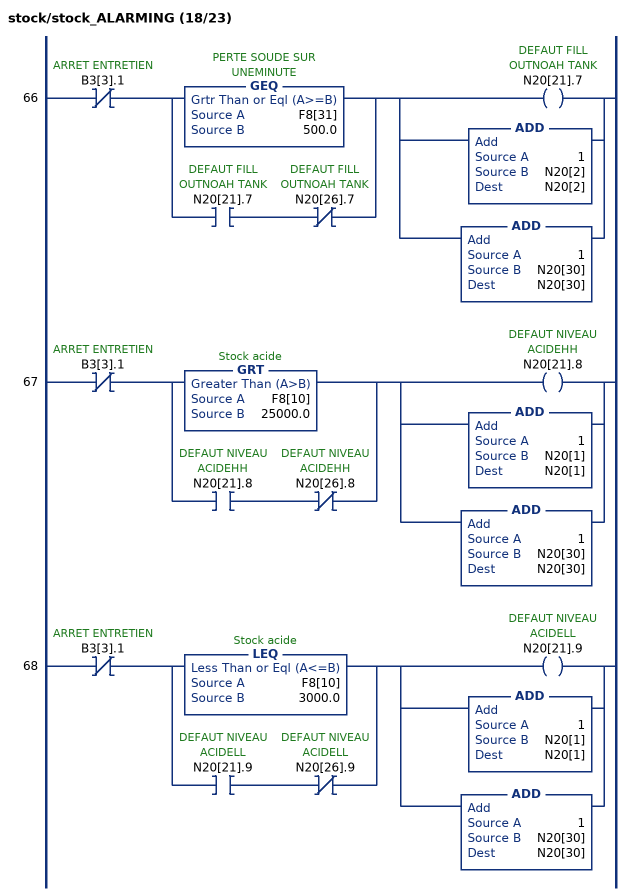
   66: XIO(B3[3].1)[GEQ(F8[31],500.0) ,XIC(N20[21].7) XIO(N20[26].7) ][OTE(N20[21].7) ,ADD(1,N20[2],N20[2]) ,ADD(1,N20[30],N20[30]) ];
   67: XIO(B3[3].1)[GRT(F8[10],25000.0) ,XIC(N20[21].8) XIO(N20[26].8) ][OTE(N20[21].8) ,ADD(1,N20[1],N20[1]) ,ADD(1,N20[30],N20[30]) ];
   68: XIO(B3[3].1)[LEQ(F8[10],3000.0) ,XIC(N20[21].9) XIO(N20[26].9) ][OTE(N20[21].9) ,ADD(1,N20[1],N20[1]) ,ADD(1,N20[30],N20[30]) ];
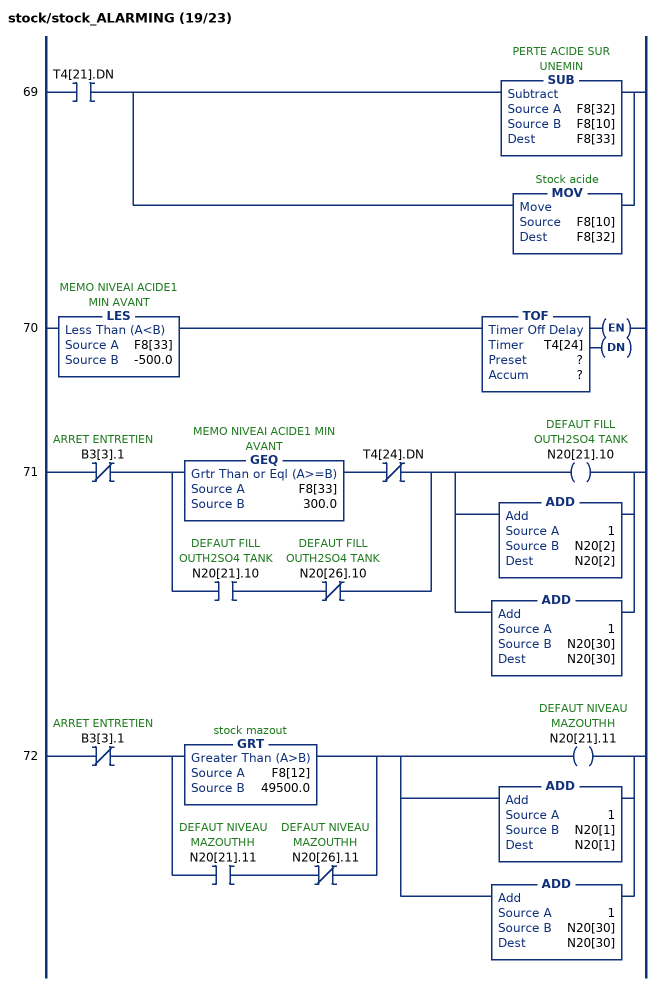
   69: XIC(T4[21].DN)[SUB(F8[32],F8[10],F8[33]) ,MOV(F8[10],F8[32]) ];
   70: LES(F8[33],-500.0)TOF(T4[24],?,?);
   71: XIO(B3[3].1)[GEQ(F8[33],300.0) XIO(T4[24].DN) ,XIC(N20[21].10) XIO(N20[26].10) ][OTE(N20[21].10) ,ADD(1,N20[2],N20[2]) ,ADD(1,N20[30],N20[30]) ];
   72: XIO(B3[3].1)[GRT(F8[12],49500.0) ,XIC(N20[21].11) XIO(N20[26].11) ][OTE(N20[21].11) ,ADD(1,N20[1],N20[1]) ,ADD(1,N20[30],N20[30]) ];
